(* LS Electric XG5000 project: 02_A+B+B-A- *)
(* PLC LSPLC *)
VAR_GLOBAL
    output_1 AT %QX0.0.1 : BOOL;
    output_2 AT %QX0.0.2 : BOOL;
    relay_1_off : BOOL;
    relay_2_off : BOOL;
    sensor_1 AT %IX0.0.1 : BOOL;
    sensor_2 AT %IX0.0.2 : BOOL;
    sensor_3 AT %IX0.0.3 : BOOL;
    sensor_4 AT %IX0.0.4 : BOOL;
END_VAR

PROGRAM NewProgram (* task: Scan Program *)
VAR_EXTERNAL
    output_1 : BOOL; (* AT %QX0.0.1 *)
    output_2 : BOOL; (* AT %QX0.0.2 *)
    relay_1_off : BOOL;
    relay_2_off : BOOL;
    sensor_1 : BOOL; (* AT %IX0.0.1 *)
    sensor_2 : BOOL; (* AT %IX0.0.2 *)
    sensor_3 : BOOL; (* AT %IX0.0.3 *)
    sensor_4 : BOOL; (* AT %IX0.0.4 *)
END_VAR

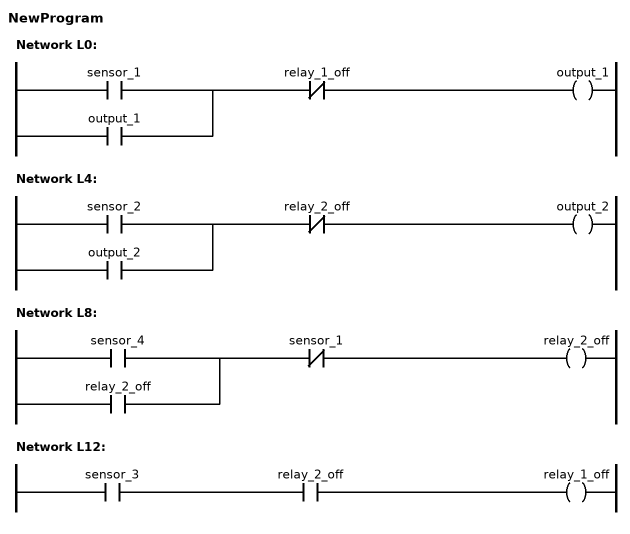
(* Rung L0 *)
output_1 := (sensor_1 OR output_1) AND NOT relay_1_off;
(* Rung L4 *)
output_2 := (sensor_2 OR output_2) AND NOT relay_2_off;
(* Rung L8 *)
relay_2_off := (sensor_4 OR relay_2_off) AND NOT sensor_1;
(* Rung L12 *)
relay_1_off := sensor_3 AND relay_2_off;
END_PROGRAM